# EPICS autosave request: iocs/tucsenIOC/iocBoot/iocTucsen/auto_settings.req
file "tucsen_settings.req",       P=$(P),  R=cam1:
file "NDStdArrays_settings.req",  P=$(P),  R=image1:
file "commonPlugin_settings.req", P=$(P)
